// TwinCAT 3 PLC project mobject_led
// Title: mobject-led
// Company: mobject
// Author: mobject-dev-team
// ProjectVersion: 0.1.1
// ProgramVersion: 3.1.4024.0
// libraries:
//   mobject-core, * (mobject)
//   Tc2_System, * (Beckhoff Automation GmbH)
// project tree:
//   Animation/ ArrayStoredAnimation.TcPOU
//   _Internal/DisplayBuffer/ I_ReadableDisplayBuffer.TcIO, I_WritableDisplayBuffer.TcIO
//   _Internal/Display/ I_Display.TcIO
//   _Internal/GraphicalElement/ I_GraphicalElement.TcIO
//   _Internal/Hardware/EL2574/DUT/ EL2574_ChannelExtendedModePdo.TcDUT, EL2574_ChannelExtendedModePdo_I.TcDUT, EL2574_ChannelExtendedModePdo_I_Status.TcDUT, EL2574_ChannelExtendedModePdo_O.TcDUT, EL2574_ChannelExtendedModePdo_O_ExtendedControl.TcDUT, EL2574_ChannelExtendedModePdo_O_ExtendedControl_Segment.TcDUT
//   _Internal/LedDevice/Interface/ I_LedDevice.TcIO
//   _Internal/LedDevice/ LedDevice.TcPOU
//   _Internal/LedDevice/Null/ NullLedDevice.TcPOU
//   _Internal/PixelFormat/ E_PixelFormat.TcDUT
//   _Internal/Pixel/ Pixel.TcDUT
//   _Internal/Scene/ I_Scene.TcIO
//   _Internal/Symbols/Interface/ I_MonoSymbol.TcIO, I_Symbol.TcIO
//   _Internal/Symbols/ Mono_16x16.TcPOU
//   DisplayBuffer/ DisplayBuffer.TcPOU
//   Hardware/EL2574/ EL2574_ChannelExtendedMode.TcPOU
//   Hardware/Matrix/ LedMatrix.TcPOU
//   / PixelColors.TcGVL
//   Scene/ Scene.TcPOU
//   Symbols/Mono_16x16/ Mono_16x16_Alarm.TcPOU, Mono_16x16_BrakeWarning.TcPOU, Mono_16x16_CircleExclamation.TcPOU, Mono_16x16_DownArrow.TcPOU, Mono_16x16_LeftArrow.TcPOU, Mono_16x16_Play.TcPOU, Mono_16x16_RightArrow.TcPOU, Mono_16x16_Smile.TcPOU, Mono_16x16_Temperature.TcPOU, Mono_16x16_TemperatureDown.TcPOU, Mono_16x16_TemperatureUp.TcPOU, Mono_16x16_UpArrow.TcPOU, Mono_16x16_User.TcPOU

// ---- _Internal/Hardware/EL2574/DUT/EL2574_ChannelExtendedModePdo.TcDUT
{attribute 'GUID' := 'B00DF5E7-F5C8-8EB2-0747-F6A66456AF18'}
{attribute 'pack_mode' := '1'}
TYPE EL2574_ChannelExtendedModePdo :
STRUCT
		{attribute 'GUID' := 'B00DF5E8-F5C8-8EB2-0747-F6A66456AF18'}
		Input AT %I* : EL2574_ChannelExtendedModePdo_I;
		{attribute 'GUID' := 'B00DF5E9-F5C8-8EB2-0747-F6A66456AF18'}
		Output AT %Q* : EL2574_ChannelExtendedModePdo_O;
	END_STRUCT
END_TYPE

// ---- _Internal/Hardware/EL2574/DUT/EL2574_ChannelExtendedModePdo_I.TcDUT
{attribute 'GUID' := 'B00DF5E8-F5C8-8EB2-0747-F6A66456AF18'}
TYPE EL2574_ChannelExtendedModePdo_I :
	STRUCT
		{attribute 'GUID' := '979B0B75-C706-0116-3B7C-F1DA38D9DB6C'}
		Status : EL2574_ChannelExtendedModePdo_I_Status;
		{attribute 'hide'}
		_reserved1 : ARRAY [1..32] OF USINT;
	END_STRUCT
END_TYPE

// ---- _Internal/Hardware/EL2574/DUT/EL2574_ChannelExtendedModePdo_I_Status.TcDUT
{attribute 'GUID' := '979B0B75-C706-0116-3B7C-F1DA38D9DB6C'}
TYPE EL2574_ChannelExtendedModePdo_I_Status :
	STRUCT
		Busy : BIT;
		Transmit : BIT;
		Send_Acknowledge : BIT;
		Update_Acknowledge : BIT;
		Command_Acknowledge : BIT;
		Command_Reject : BIT;
		 {attribute 'hide'}
		_reserved1 : BIT;
		 {attribute 'hide'}
		_reserved2 : BIT;
		 {attribute 'hide'}
		_reserved3 : BIT;
		 {attribute 'hide'}
		_reserved4 : BIT;
		Warning : BIT;
		Error : BIT;
		 {attribute 'hide'}
		_reserved5 : BIT;
		 {attribute 'hide'}
		_reserved6 : BIT;
		 {attribute 'GUID' := '18071995-0000-0000-0000-000000000010}
		Input_Cycle_Counter_Bit0 : BIT;
		 {attribute 'GUID' := '18071995-0000-0000-0000-000000000010}
		Input_Cycle_Counter_Bit1 : BIT;
	END_STRUCT
END_TYPE

// ---- _Internal/Hardware/EL2574/DUT/EL2574_ChannelExtendedModePdo_O.TcDUT
{attribute 'GUID' := 'B00DF5E9-F5C8-8EB2-0747-F6A66456AF18'}
{attribute 'pack_mode' := '1'}
TYPE EL2574_ChannelExtendedModePdo_O :
	STRUCT
		 {attribute 'GUID' := 'FCFFC25C-7C92-C549-757B-D5CF9395F3F6'}
		ExtendedControl : EL2574_ChannelExtendedModePdo_O_ExtendedControl;
	END_STRUCT
END_TYPE

// ---- _Internal/Hardware/EL2574/DUT/EL2574_ChannelExtendedModePdo_O_ExtendedControl.TcDUT
{attribute 'GUID' := 'FCFFC25C-7C92-C549-757B-D5CF9395F3F6'}
{attribute 'pack_mode' := '1'}
TYPE EL2574_ChannelExtendedModePdo_O_ExtendedControl :
	STRUCT
		Execute : BIT;
		Send : BIT;
		Update : BIT;
		Write : BIT;
		 {attribute 'hide'}
		_reserved1 : BIT;
		 {attribute 'hide'}
		_reserved2 : BIT;
		 {attribute 'hide'}
		_reserved3 : BIT;
		 {attribute 'hide'}
		_reserved4 : BIT;
		Index : USINT;
		 {attribute 'GUID' := 'C34ECFC1-C235-2097-8F87-A8742B490E4F'}
		Segment : EL2574_ChannelExtendedModePdo_O_ExtendedControl_Segment;
	END_STRUCT
END_TYPE

// ---- _Internal/Hardware/EL2574/DUT/EL2574_ChannelExtendedModePdo_O_ExtendedControl_Segment.TcDUT
{attribute 'GUID' := 'C34ECFC1-C235-2097-8F87-A8742B490E4F'}
TYPE EL2574_ChannelExtendedModePdo_O_ExtendedControl_Segment :
	STRUCT
		Element_0 : UDINT;
		Element_1 : UDINT;
		Element_2 : UDINT;
		Element_3 : UDINT;
		Element_4 : UDINT;
		Element_5 : UDINT;
		Element_6 : UDINT;
		Element_7 : UDINT;
	END_STRUCT
END_TYPE

// ---- _Internal/PixelFormat/E_PixelFormat.TcDUT
{attribute 'qualified_only'}
{attribute 'strict'}
TYPE E_PixelFormat :
(
	RRGGBBAA,
	AARRGGBB,
	xxRRGGBB
);
END_TYPE

// ---- _Internal/Pixel/Pixel.TcDUT
TYPE Pixel : UDINT; END_TYPE

// ---- PixelColors.TcGVL
{attribute 'qualified_only'}
VAR_GLOBAL CONSTANT;
	RED : Pixel := 16#FF0000FF;
	GREEN : Pixel := 16#00FF00FF;
	BLUE : Pixel := 16#0000FFFF;
	YELLOW : Pixel := 16#FFFF00FF;
	BLACK : Pixel := 16#000000FF;
	WHITE : Pixel := 16#FFFFFFF;
	PURPLE : Pixel := 16#800080FF;
	ORANGE : Pixel := 16#FFA500FF;
	GREY : Pixel := 16#808080FF;
	TEAL : Pixel := 16#008080FF;
	CYAN : Pixel := 16#00FFFFF;
	MAGENTA : Pixel := 16#FF00FFFF;
	LIME : Pixel := 16#00FF00FF;
	PINK : Pixel := 16#FFC0CBFF;
	BROWN : Pixel := 16#A52A2AFF;
	NAVY : Pixel := 16#000080FF;
	OLIVE : Pixel := 16#808000FF;
	MAROON : Pixel := 16#800000FF;
	AQUA : Pixel := 16#00FFFFF;
END_VAR

// ---- _Internal/DisplayBuffer/I_ReadableDisplayBuffer.TcIO
INTERFACE I_ReadableDisplayBuffer

METHOD PUBLIC TryReadPixel : BOOL;
VAR_INPUT
	X : DINT;
	Y : DINT;
	Pixel : REFERENCE TO Pixel;
END_VAR
END_METHOD

END_INTERFACE

// ---- _Internal/DisplayBuffer/I_WritableDisplayBuffer.TcIO
INTERFACE I_WritableDisplayBuffer

METHOD PUBLIC SetPixel
VAR_INPUT
	X : DINT;
	Y : DINT;
	Pixel : Pixel;
END_VAR
END_METHOD

END_INTERFACE

// ---- _Internal/Display/I_Display.TcIO
INTERFACE I_Display

METHOD PUBLIC UpdateFrom
VAR_INPUT
	Source : I_ReadableDisplayBuffer;
END_VAR
END_METHOD

END_INTERFACE

// ---- _Internal/GraphicalElement/I_GraphicalElement.TcIO
INTERFACE I_GraphicalElement

METHOD PUBLIC RenderTo
VAR_INPUT
	Destination : I_WritableDisplayBuffer;
END_VAR
END_METHOD

METHOD PUBLIC Update
VAR_INPUT
	DeltaTimeInMs : UDINT;
END_VAR
END_METHOD

END_INTERFACE

// ---- _Internal/LedDevice/Interface/I_LedDevice.TcIO
INTERFACE I_LedDevice EXTENDS I_Display

METHOD PUBLIC ConnectTo
VAR_INPUT
	LedDevice : I_LedDevice;
END_VAR
END_METHOD

METHOD PUBLIC ResetPixelPointer
VAR_INPUT
END_VAR
END_METHOD

METHOD PUBLIC TryGetNextPixel : BOOL
VAR_INPUT
	Destination : REFERENCE TO Pixel;
END_VAR
END_METHOD

METHOD PUBLIC UpdateFrom
VAR_INPUT
	Source : I_ReadableDisplayBuffer;
END_VAR
END_METHOD

END_INTERFACE

// ---- _Internal/Scene/I_Scene.TcIO
INTERFACE I_Scene EXTENDS I_GraphicalElement

METHOD Clear
VAR_INPUT
END_VAR
END_METHOD

METHOD PUBLIC TryAddElement
VAR_INPUT
	GraphicalElement : I_GraphicalElement;
END_VAR
END_METHOD

METHOD PUBLIC TryRemoveElement
VAR_INPUT
	GraphicalElement : I_GraphicalElement;
END_VAR
END_METHOD

END_INTERFACE

// ---- _Internal/Symbols/Interface/I_MonoSymbol.TcIO
INTERFACE I_MonoSymbol EXTENDS I_Symbol

PROPERTY PUBLIC BackgroundColor : Pixel
GET
END_GET
SET
END_SET
END_PROPERTY

PROPERTY PUBLIC ForgroundColor : Pixel
GET
END_GET
SET
END_SET
END_PROPERTY

METHOD PUBLIC InvertColor
VAR_INPUT
END_VAR
END_METHOD

END_INTERFACE

// ---- _Internal/Symbols/Interface/I_Symbol.TcIO
INTERFACE I_Symbol EXTENDS I_GraphicalElement

PROPERTY PUBLIC FlipX : BOOL
GET
END_GET
SET
END_SET
END_PROPERTY

PROPERTY PUBLIC FlipY : BOOL
GET
END_GET
SET
END_SET
END_PROPERTY

PROPERTY PUBLIC Rotation : UINT
GET
END_GET
SET
END_SET
END_PROPERTY

END_INTERFACE

// ---- Animation/ArrayStoredAnimation.TcPOU
{attribute 'linkalways'} 
{attribute 'no_explicit_call' := 'This FB is a CLASS and must be accessed using methods or properties'}
{attribute 'enable_dynamic_creation'}
FUNCTION_BLOCK ArrayStoredAnimation IMPLEMENTS I_GraphicalElement
VAR
	// setup
	_width : UDINT;
	_height : UDINT;
	
	// buffer
	expectedFrameSizeInBytes : UDINT;
	frameCount : UDINT;
	pAnimationFrameData : POINTER TO Pixel;
	nAnimationFrameData : UDINT;
	
	// animation
	currentFrameIndex : UDINT;
	pCurrentFrame : POINTER TO Pixel;
	elapsedTimeInMs : UDINT;
END_VAR

METHOD FB_exit : BOOL
VAR_INPUT
	bInCopyCode : BOOL; // if TRUE, the exit method is called for exiting an instance that is copied afterwards (online change).
END_VAR
IF bInCopyCode THEN
	RETURN;
END_IF

IF pAnimationFrameData = 0 THEN
	RETURN;
END_IF

__DELETE(pAnimationFrameData);
END_METHOD

METHOD FB_init : BOOL
VAR_INPUT
	bInitRetains : BOOL; // if TRUE, the retain variables are initialized (warm start / cold start)
	bInCopyCode : BOOL;  // if TRUE, the instance afterwards gets moved into the copy code (online change)
	Width : UDINT;
	Height : UDINT;
END_VAR
_width := Width;
_height := Height;
UpdateExpectedFrameSizeInBytes();
END_METHOD

PROPERTY PUBLIC Height : UDINT
GET
Height := _height;
END_GET
END_PROPERTY

METHOD PUBLIC RenderTo
VAR_INPUT
	Destination : I_WritableDisplayBuffer;
END_VAR
// needs implementation

//IF X > _width THEN
//	RETURN;
//END_IF

//IF Y > _height THEN
//	RETURN;
//END_IF

//IF frameCount = 0 THEN
//	RETURN;
//END_IF

//offset := (y * width) + x;
//Destination := pCurrentFrame[offset];
//GetPixel := TRUE;
END_METHOD

METHOD PUBLIC Reset : BOOL
VAR_INPUT
END_VAR
Reset := TryGoToFrame(0);
END_METHOD

METHOD PRIVATE ResetAnimation
VAR_INPUT
END_VAR
currentFrameIndex := 0;
pCurrentFrame := pAnimationFrameData;
END_METHOD

METHOD PUBLIC TryAddFrame : BOOL
VAR_INPUT
	FrameDataArray : ANY;
END_VAR
VAR
	newFrameCount : UDINT;
	newAnimationDataSize : UDINT;
	pNewAnimationFrameData : POINTER TO pixel;
	pNewFrameStart : POINTER TO pixel; 
END_VAR
IF FrameDataArray.pValue = 0 THEN
	RETURN;
END_IF

IF FrameDataArray.diSize = 0 THEN
	RETURN;
END_IF

IF FrameDataArray.diSize <> expectedFrameSizeInBytes THEN
	RETURN;
END_IF

// setup the new buffer (one frame bigger than previous)
newFrameCount := frameCount + 1;
newAnimationDataSize := expectedFrameSizeInBytes * newFrameCount;
pNewAnimationFrameData := __NEW(BYTE, newAnimationDataSize);

// copy the old data across if available;
IF nAnimationFrameData > 0 THEN
	memcpy(pNewAnimationFrameData, pAnimationFrameData, nAnimationFrameData); 
	__DELETE(pAnimationFrameData);
	pAnimationFrameData := 0;
	nAnimationFrameData := 0;
END_IF

// copy the supplied frame data to the end of the new buffer.
pNewFrameStart := pNewAnimationFrameData + (frameCount * expectedFrameSizeInBytes);
memcpy(pNewFrameStart, FrameDataArray.pValue, FrameDataArray.diSize); 

// update internal values to the new values.
pAnimationFrameData := pNewAnimationFrameData;
nAnimationFrameData := newAnimationDataSize;
frameCount := newFrameCount;

// reset animation
ResetAnimation();

// success
TryAddFrame := TRUE;
END_METHOD

METHOD PUBLIC TryGoToFrame : BOOL
VAR_INPUT
	AnimationFrameIndex : UDINT;
END_VAR
IF frameCount = 0 THEN 
	RETURN;
END_IF

IF AnimationFrameIndex > frameCount THEN
	RETURN;
END_IF

currentFrameIndex := AnimationFrameIndex;
pCurrentFrame := pAnimationFrameData + (currentFrameIndex * expectedFrameSizeInBytes);
TryGoToFrame := TRUE;
END_METHOD

METHOD PUBLIC TryGoToNextFrame : BOOL
VAR_INPUT
END_VAR
TryGoToNextFrame := TryGoToFrame(currentFrameIndex + 1);
END_METHOD

METHOD PUBLIC Update
VAR_INPUT
	DeltaTimeInMs : UDINT;
END_VAR
// not implemented
END_METHOD

METHOD PRIVATE UpdateExpectedFrameSizeInBytes
VAR
	tempPixel : Pixel;
END_VAR
expectedFrameSizeInBytes := SIZEOF(tempPixel) * this^._width * this^._height;
END_METHOD

PROPERTY PUBLIC Width : UDINT
GET
Width := _width;
END_GET
END_PROPERTY

END_FUNCTION_BLOCK

// ---- _Internal/LedDevice/LedDevice.TcPOU
{attribute 'linkalways'} 
{attribute 'no_explicit_call' := 'This FB is a CLASS and must be accessed using methods or properties'}
{attribute 'enable_dynamic_creation'}
FUNCTION_BLOCK ABSTRACT LedDevice IMPLEMENTS I_LedDevice
VAR
	// using the null object pattern so that you no longer need to check to see if next is <> 0
	nullLedDevice : NullLedDevice;
	next : I_LedDevice := NullLedDevice;
	allPixelsSerialized : BOOL;
	_requiredPixelFormat : E_PixelFormat := E_PixelFormat.AARRGGBB;
END_VAR

METHOD PUBLIC ConnectTo
VAR_INPUT
	LedDevice : I_LedDevice;
END_VAR
IF LedDevice = 0  THEN
	next := nullLedDevice;
END_IF

IF LedDevice = next THEN
	RETURN;
END_IF

next := LedDevice;
END_METHOD

METHOD PROTECTED Convert_RGBA_To_RequiredPixelFormat : Pixel
VAR_INPUT
	Input : Pixel;
END_VAR
CASE _requiredPixelFormat OF
	E_PixelFormat.RRGGBBAA :
		Convert_RGBA_To_RequiredPixelFormat := Input;
		
	E_PixelFormat.AARRGGBB, 
	E_PixelFormat.xxRRGGBB :
		Convert_RGBA_To_RequiredPixelFormat := ROR(Input,8) ; 
END_CASE
END_METHOD

PROPERTY PUBLIC NextDevice : I_LedDevice
GET
NextDevice := next;
END_GET
END_PROPERTY

METHOD PROTECTED ABSTRACT OnResetPixelPointer
VAR_INPUT
END_VAR
// a serializer will be instructed to reset it's own pixel tracking here. 
// this indicates that the next time OnTryGetNextPixel is called, the first pixel must be returned;
END_METHOD

METHOD PROTECTED ABSTRACT OnTryGetNextPixel : BOOL
VAR_INPUT
	Destination : REFERENCE TO Pixel;
END_VAR
// a serializer must keep track of it's own next pixel and set the destination, and return true when called.  
// if there are no further pixels you must return false
END_METHOD

METHOD PROTECTED ABSTRACT OnUpdateFrom
VAR_INPUT
	Source : I_ReadableDisplayBuffer;
END_VAR
END_METHOD

PROPERTY PUBLIC RequiredPixelFormat : E_PixelFormat
GET
RequiredPixelFormat := _requiredPixelFormat;
END_GET
SET
_requiredPixelFormat := RequiredPixelFormat;
END_SET
END_PROPERTY

METHOD PUBLIC ResetPixelPointer
VAR_INPUT
END_VAR
OnResetPixelPointer();
allPixelsSerialized := FALSE;
NextDevice.ResetPixelPointer();
END_METHOD

METHOD PUBLIC TryGetNextPixel : BOOL
VAR_INPUT
	Destination : REFERENCE TO Pixel;
END_VAR
IF allPixelsSerialized THEN
	TryGetNextPixel := NextDevice.TryGetNextPixel(Destination);
	RETURN;
END_IF

IF OnTryGetNextPixel(Destination) THEN
	TryGetNextPixel := TRUE;
	RETURN;
END_IF

allPixelsSerialized := TRUE;
TryGetNextPixel := NextDevice.TryGetNextPixel(Destination);
END_METHOD

METHOD PUBLIC UpdateFrom
VAR_INPUT
	Source : I_ReadableDisplayBuffer;
END_VAR
IF Source = 0 THEN
	RETURN;
END_IF

OnUpdateFrom(Source);
END_METHOD

END_FUNCTION_BLOCK

// ---- _Internal/LedDevice/Null/NullLedDevice.TcPOU
{attribute 'linkalways'} 
{attribute 'no_explicit_call' := 'This FB is a CLASS and must be accessed using methods or properties'}
{attribute 'enable_dynamic_creation'}
FUNCTION_BLOCK NullLedDevice IMPLEMENTS I_LedDevice
VAR
END_VAR

METHOD PUBLIC ConnectTo
VAR_INPUT
	LedDevice : I_LedDevice;
END_VAR
// no code here..
END_METHOD

METHOD PUBLIC ResetPixelPointer
VAR_INPUT
END_VAR
// no code here..
END_METHOD

METHOD PUBLIC TryGetNextPixel : BOOL
VAR_INPUT
	Destination : REFERENCE TO Pixel;
END_VAR
TryGetNextPixel := FALSE;
END_METHOD

METHOD PUBLIC UpdateFrom
VAR_INPUT
	Source : I_ReadableDisplayBuffer;
END_VAR
// no code here..
END_METHOD

END_FUNCTION_BLOCK

// ---- _Internal/Symbols/Mono_16x16.TcPOU
{attribute 'linkalways'} 
{attribute 'no_explicit_call' := 'This FB is a CLASS and must be accessed using methods or properties'}
{attribute 'enable_dynamic_creation'}
FUNCTION_BLOCK ABSTRACT Mono_16x16 IMPLEMENTS I_MonoSymbol
VAR
	_x : DINT;
	_y : DINT;
	_flipX : BOOL;
	_flipY : BOOL;
	_rotation : UINT;
	_forgroundColor : Pixel := WHITE;
	_backgroundColor : Pixel := TRANSPARENT;
END_VAR
VAR CONSTANT
	SYMBOL_WIDTH : UDINT := 16;
	SYMBOL_HEIGHT : UDINT := 16;
	WHITE : Pixel := 16#FFFFFFFF;
	TRANSPARENT : Pixel := 16#00000000;
END_VAR

PROPERTY PUBLIC BackgroundColor : Pixel
GET
BackgroundColor := _backgroundColor;
END_GET
SET
_backgroundColor := BackgroundColor;
END_SET
END_PROPERTY

METHOD FB_init : BOOL
VAR_INPUT
	bInitRetains : BOOL; // if TRUE, the retain variables are initialized (warm start / cold start)
	bInCopyCode : BOOL;  // if TRUE, the instance afterwards gets moved into the copy code (online change)
	Forground : Pixel;
	Background : Pixel;
END_VAR
_forgroundColor := Forground;
_backgroundColor := Background;
END_METHOD

PROPERTY PUBLIC FlipX : BOOL
GET
FlipX := _flipX;
END_GET
SET
_flipX := FlipX;
END_SET
END_PROPERTY

PROPERTY PUBLIC FlipY : BOOL
GET
FlipY := _flipY;
END_GET
SET
_flipY := FlipY;
END_SET
END_PROPERTY

PROPERTY PUBLIC ForgroundColor : Pixel
GET
ForgroundColor := _forgroundColor;
END_GET
SET
_forgroundColor := ForgroundColor;
END_SET
END_PROPERTY

PROPERTY PUBLIC Height : UDINT
GET
Height := SYMBOL_HEIGHT;
END_GET
END_PROPERTY

METHOD PUBLIC InvertColor
VAR_INPUT
END_VAR
END_METHOD

PROPERTY PROTECTED ABSTRACT Pixels : REFERENCE TO ARRAY [0..255] of BYTE
GET
END_GET
END_PROPERTY

METHOD PUBLIC RenderTo
VAR_INPUT
	Destination : I_WritableDisplayBuffer;
END_VAR
VAR
	row : UDINT;
	column : UDINT;
	newRow : UDINT;
	newColumn : UDINT;
	pixelOffset : UDINT;
	destinationX : DINT;
	destinationY : DINT;
END_VAR
FOR row := 0 TO SYMBOL_HEIGHT - 1 DO
	FOR column := 0 TO SYMBOL_WIDTH - 1 DO

		CASE _rotation OF
			
			0:
				newColumn := column;
				newRow := row;
			90:
				newColumn := SYMBOL_HEIGHT - 1 - row;
				newRow := column;
			180:
				newColumn := SYMBOL_WIDTH - 1 - column;
				newRow := SYMBOL_HEIGHT - 1 - row;
			270:
				newColumn := row;
				newRow := SYMBOL_WIDTH - 1 - column;
			
		END_CASE

		IF _flipX THEN
			newColumn := SYMBOL_WIDTH - 1 - newColumn;
		END_IF

		IF _flipY THEN
			newRow := SYMBOL_HEIGHT - 1 - newRow;
		END_IF

		pixelOffset := (newRow * SYMBOL_WIDTH) + newColumn;
		destinationX := UDINT_TO_DINT(column) + _x;
		destinationY := UDINT_TO_DINT(row) + _y;
		
		IF Pixels[pixelOffset] = 0 THEN
			Destination.SetPixel(destinationX, destinationY, _backgroundColor);
		ELSE
			Destination.SetPixel(destinationX, destinationY, _forgroundColor);
		END_IF

	END_FOR
END_FOR
END_METHOD

PROPERTY PUBLIC Rotation : UINT
GET
Rotation := _rotation;
END_GET
SET
_rotation := Rotation;
END_SET
END_PROPERTY

METHOD PUBLIC Update
VAR_INPUT
	DeltaTimeInMs : UDINT;
END_VAR
// not required for static symbols
END_METHOD

PROPERTY PUBLIC Width : UDINT
GET
Width := SYMBOL_WIDTH;
END_GET
END_PROPERTY

PROPERTY PUBLIC X : DINT
GET
X := _x;
END_GET
SET
_x := X;
END_SET
END_PROPERTY

PROPERTY PUBLIC Y : DINT
GET
Y := _y;
END_GET
SET
_y := Y;
END_SET
END_PROPERTY

END_FUNCTION_BLOCK

// ---- DisplayBuffer/DisplayBuffer.TcPOU
{attribute 'linkalways'} 
{attribute 'no_explicit_call' := 'This FB is a CLASS and must be accessed using methods or properties'}
{attribute 'enable_dynamic_creation'}
FUNCTION_BLOCK DisplayBuffer IMPLEMENTS I_WritableDisplayBuffer, I_ReadableDisplayBuffer
VAR
	// setup
	_width : UDINT;
	_height : UDINT;
	
	// buffer
	displayBufferSize : UDINT;
	pDisplayBuffer : POINTER TO Pixel;
END_VAR

METHOD PUBLIC Clear
VAR_INPUT
END_VAR
IF pDisplayBuffer = 0 THEN
	RETURN;
END_IF

memset(pDisplayBuffer, 0, displayBufferSize);
END_METHOD

METHOD PRIVATE CreateDisplayBuffer
VAR
	tempPixel : Pixel;
END_VAR
displayBufferSize := _width * _height * SIZEOF(tempPixel);
pDisplayBuffer := __NEW(BYTE, displayBufferSize);
memset(pDisplayBuffer, 0, displayBufferSize);
END_METHOD

METHOD FB_exit : BOOL
VAR_INPUT
	bInCopyCode : BOOL; // if TRUE, the exit method is called for exiting an instance that is copied afterwards (online change).
END_VAR
IF bInCopyCode THEN
	RETURN;
END_IF

IF pDisplayBuffer = 0 THEN
	RETURN;
END_IF

__DELETE(pDisplayBuffer);
END_METHOD

METHOD FB_init : BOOL
VAR_INPUT
	bInitRetains : BOOL; // if TRUE, the retain variables are initialized (warm start / cold start)
	bInCopyCode : BOOL;  // if TRUE, the instance afterwards gets moved into the copy code (online change)
	Width : UDINT;
	Height : UDINT;
END_VAR
_width := Width;
_height := Height;
CreateDisplayBuffer();
END_METHOD

PROPERTY PUBLIC Height : UDINT
GET
Height := _height;
END_GET
END_PROPERTY

METHOD PUBLIC SendTo
VAR_INPUT
	Display : I_Display;
END_VAR
Display.UpdateFrom(this^);
END_METHOD

METHOD PUBLIC SetPixel
VAR_INPUT
	X : DINT;
	Y : DINT;
	Pixel : Pixel;
END_VAR
VAR
	xAsUdint : UDINT;
	yAsUdint : UDINT;
	offset : UDINT;
END_VAR
IF X < 0 THEN
	RETURN;
END_IF

IF Y < 0 THEN
	RETURN;
END_IF

xAsUdint := DINT_TO_UDINT(X);
yAsUdint := DINT_TO_UDINT(Y);

IF xAsUdint >= _width THEN
	RETURN;
END_IF

IF yAsUdint >= _height THEN
	RETURN;
END_IF


offset := (yAsUdint * _width) + xAsUdint;

IF offset = 176 THEN
			offset := offset;
		END_IF

		
pDisplayBuffer[offset] := Pixel;
END_METHOD

METHOD PUBLIC TryCopyTo : BOOL
VAR_INPUT
	Destination : ANY;
END_VAR
IF DINT_TO_UDINT(Destination.diSize) < displayBufferSize THEN
	RETURN;
END_IF

memcpy(Destination.pValue, pDisplayBuffer, displayBufferSize);
TryCopyTo := true;
END_METHOD

METHOD PUBLIC TryReadPixel : BOOL;
VAR_INPUT
	X : DINT;
	Y : DINT;
	Pixel : REFERENCE TO Pixel;
END_VAR
VAR
	xAsUdint : UDINT;
	yAsUdint : UDINT;
	offset : UDINT;
END_VAR
IF X < 0 THEN
	RETURN;
END_IF

IF Y < 0 THEN
	RETURN;
END_IF

xAsUdint := DINT_TO_UDINT(X);
yAsUdint := DINT_TO_UDINT(Y);

IF xAsUdint >= _width THEN
	RETURN;
END_IF

IF yAsUdint >= _height THEN
	RETURN;
END_IF

offset := (yAsUdint * _width) + xAsUdint;
Pixel := pDisplayBuffer[offset];
TryReadPixel := TRUE;
END_METHOD

PROPERTY PUBLIC Width : UDINT
GET
Width := _width;
END_GET
END_PROPERTY

END_FUNCTION_BLOCK

// ---- Hardware/EL2574/EL2574_ChannelExtendedMode.TcPOU
{attribute 'linkalways'} 
{attribute 'no_explicit_call' := 'This FB is a CLASS and must be accessed using methods or properties'}
{attribute 'enable_dynamic_creation'}
FUNCTION_BLOCK EL2574_ChannelExtendedMode
VAR
	pdo : EL2574_ChannelExtendedModePdo;
	nullLedDevice : NullLedDevice;
	connectedTo : I_LedDevice := NullLedDevice;
	
	totalPixels : UDINT;
	sendBuffer : ARRAY [0..MAX_PIXELS - 1] OF UDINT;
	sendSegmentCount : USINT;
	currentSegment : USINT;
	state : (IDLE, INITIALIZING, SEND_SEGMENT, TRIGGER_FRAME_SEND, WAIT_FOR_FRAME_SEND_COMPLETE, ERROR);
END_VAR
VAR CONSTANT
	MAX_PIXELS : UDINT := 2048;
END_VAR

METHOD PUBLIC ConnectTo
VAR_INPUT
	LedDevice : I_LedDevice;
END_VAR
IF LedDevice = 0  THEN
	connectedTo := nullLedDevice;
END_IF

IF LedDevice = connectedTo THEN
	RETURN;
END_IF

connectedTo := LedDevice;
END_METHOD

METHOD PUBLIC CyclicCall
VAR_INPUT
END_VAR
VAR
	totalSegments : UDINT;
	currentPixel : UDINT;
	i : UDINT;
END_VAR
CASE state OF
	
	IDLE : 

		IF connectedTo = 0 THEN
			RETURN;
		END_IF
		
		connectedTo.ResetPixelPointer();
		currentPixel := 0;
		
		// fetch the buffer
		WHILE connectedTo.TryGetNextPixel(sendBuffer[currentPixel]) DO
			currentPixel := currentPixel + 1;
		END_WHILE
		
		totalPixels := currentPixel;
		
		// reset the remainder of the buffer
		FOR i := currentPixel + 1 TO MAX_PIXELS -1 DO 
			sendBuffer[i] := 16#0;
		END_FOR
		
		state := INITIALIZING;
		
	ERROR : RETURN;
	
	INITIALIZING :
	
		// initialize local variables
		currentSegment := 0;
		totalSegments := totalPixels / 8;
		sendSegmentCount := UDINT_TO_USINT(totalSegments);
	
		// reset the card to a known state 
		pdo.Output.ExtendedControl.Index := 0;
		pdo.Output.ExtendedControl.Send := FALSE;
		pdo.Output.ExtendedControl.Update := FALSE;
		pdo.Output.ExtendedControl.Write := FALSE;
		pdo.Output.ExtendedControl.Segment.Element_0 := 0;
		pdo.Output.ExtendedControl.Segment.Element_1 := 0;
		pdo.Output.ExtendedControl.Segment.Element_2 := 0;
		pdo.Output.ExtendedControl.Segment.Element_3 := 0;
		pdo.Output.ExtendedControl.Segment.Element_4 := 0;
		pdo.Output.ExtendedControl.Segment.Element_5 := 0;
		pdo.Output.ExtendedControl.Segment.Element_6 := 0;
		pdo.Output.ExtendedControl.Segment.Element_7 := 0;
		
		// start sending....
		state := SEND_SEGMENT;

	SEND_SEGMENT :
		
		pdo.Output.ExtendedControl.Index := currentSegment;
		pdo.Output.ExtendedControl.Segment.Element_0 := sendBuffer[currentSegment * 8 + 0];
		pdo.Output.ExtendedControl.Segment.Element_1 := sendBuffer[currentSegment * 8 + 1];
		pdo.Output.ExtendedControl.Segment.Element_2 := sendBuffer[currentSegment * 8 + 2];
		pdo.Output.ExtendedControl.Segment.Element_3 := sendBuffer[currentSegment * 8 + 3];
		pdo.Output.ExtendedControl.Segment.Element_4 := sendBuffer[currentSegment * 8 + 4];
		pdo.Output.ExtendedControl.Segment.Element_5 := sendBuffer[currentSegment * 8 + 5];
		pdo.Output.ExtendedControl.Segment.Element_6 := sendBuffer[currentSegment * 8 + 6];
		pdo.Output.ExtendedControl.Segment.Element_7 := sendBuffer[currentSegment * 8 + 7];
		pdo.Output.ExtendedControl.Write := TRUE;
		pdo.Output.ExtendedControl.Execute := NOT pdo.Output.ExtendedControl.Execute;
		
		IF currentSegment = sendSegmentCount THEN
			state := TRIGGER_FRAME_SEND;
		ELSE
			currentSegment := currentSegment + 1;
		END_IF
		
	TRIGGER_FRAME_SEND : 
	
		pdo.Output.ExtendedControl.Write := FALSE;
		pdo.Output.ExtendedControl.Update := TRUE;
		pdo.Output.ExtendedControl.Send := TRUE;
		pdo.Output.ExtendedControl.Execute := NOT pdo.Output.ExtendedControl.Execute;
		
		state := WAIT_FOR_FRAME_SEND_COMPLETE;
		
	WAIT_FOR_FRAME_SEND_COMPLETE:
	
		IF NOT pdo.Input.Status.Busy THEN
			pdo.Output.ExtendedControl.Update := FALSE;
			pdo.Output.ExtendedControl.Send := FALSE;
			state := IDLE;
		END_IF

		
END_CASE
END_METHOD

PROPERTY PUBLIC HasError : BOOL
GET
HasError := state = Error;
END_GET
END_PROPERTY

PROPERTY PUBLIC IsBusy : BOOL
GET
IsBusy := not(state = IDLE or_else state = ERROR);
END_GET
END_PROPERTY

END_FUNCTION_BLOCK

// ---- Hardware/Matrix/LedMatrix.TcPOU
{attribute 'linkalways'} 
{attribute 'no_explicit_call' := 'This FB is a CLASS and must be accessed using methods or properties'}
{attribute 'enable_dynamic_creation'}
FUNCTION_BLOCK LedMatrix EXTENDS LedDevice
VAR
	// setup
	height : UDINT;
	width : UDINT;
	x : DINT;
	y : DINT;
	flipX : BOOL;
	flipY : BOOL;
	rotation : UINT;
	
	// buffer
	pixelBufferSize : UDINT;
	pPixelBuffer : POINTER TO Pixel;
	
	// serializer
	nextPixel : UDINT;
END_VAR

METHOD PRIVATE CreatePixelBuffer
VAR
	tempPixel : Pixel;
END_VAR
pixelBufferSize := width * height * SIZEOF(tempPixel);
pPixelBuffer := __NEW(BYTE, pixelBufferSize);
memset(pPixelBuffer, 0, pixelBufferSize);
END_METHOD

METHOD FB_exit : BOOL
VAR_INPUT
	bInCopyCode : BOOL; // if TRUE, the exit method is called for exiting an instance that is copied afterwards (online change).
END_VAR
IF bInCopyCode THEN
	RETURN;
END_IF

IF pPixelBuffer = 0 THEN
	RETURN;
END_IF

__DELETE(pPixelBuffer);
END_METHOD

METHOD FB_init : BOOL
VAR_INPUT
	bInitRetains : BOOL; // if TRUE, the retain variables are initialized (warm start / cold start)
	bInCopyCode : BOOL;  // if TRUE, the instance afterwards gets moved into the copy code (online change)
	Height : UDINT;
	Width : UDINT;
	X : UDINT;
	Y : UDINT;
	FlipX : BOOL;
	FlipY : BOOL;
	Rotation : UINT;
END_VAR
THIS^.height := Height;
THIS^.width := Width;
THIS^.x := X;
THIS^.y := Y;
THIS^.flipX := FlipX;
THIS^.flipY := FlipY;
THIS^.rotation := Rotation;

CreatePixelBuffer();
END_METHOD

METHOD PROTECTED OnResetPixelPointer
VAR_INPUT
END_VAR
nextPixel := 0;
END_METHOD

METHOD PROTECTED OnTryGetNextPixel : BOOL
VAR_INPUT
	Destination : REFERENCE TO Pixel;
END_VAR
IF nextPixel > pixelBufferSize THEN
	OnTryGetNextPixel := FALSE;
	RETURN;
END_IF

IF pixelBufferSize = 0 THEN
	RETURN;
END_IF

Destination := pPixelBuffer[nextPixel];
nextPixel := nextPixel + 1;
OnTryGetNextPixel := TRUE;
END_METHOD

METHOD PROTECTED OnUpdateFrom
VAR_INPUT
	Source : I_ReadableDisplayBuffer;
END_VAR
VAR
	row : UDINT;
	column : UDINT;
	newRow : UDINT;
	newColumn : UDINT;
	destinationX : DINT;
	destinationY : DINT;
	index: UDINT;
	pixelValue : PIXEL;
END_VAR
FOR row := 0 TO height - 1 DO
	FOR column := 0 TO width - 1 DO
		
		// calculate the index of our own buffer which represents the current col and row
		IF row MOD 2 = 1 THEN
			// on an odd row the direction is reversed.
			index := row * width + ((width - 1) - column);
		ELSE
			index := row * width + column;
		END_IF
		
		CASE rotation OF
			
			0:
				newColumn := column;
				newRow := row;
			90:
				newColumn := height - 1 - row;
				newRow := column;
			180:
				newColumn := width - 1 - column;
				newRow := height - 1 - row;
			270:
				newColumn := row;
				newRow := width - 1 - column;
			
		END_CASE

		IF flipX THEN
			newColumn := width - 1 - newColumn;
		END_IF

		IF flipY THEN
			newRow := height - 1 - newRow;
		END_IF

		destinationX := UDINT_TO_DINT(newColumn) + x;
		destinationY := UDINT_TO_DINT(newRow) + y;
		
		IF NOT Source.TryReadPixel(destinationX, destinationY, pixelValue) THEN
			pPixelBuffer[index] := 16#00000000;
			RETURN;
		END_IF
		
		pPixelBuffer[index] := THIS^.Convert_RGBA_To_RequiredPixelFormat(pixelValue);

	END_FOR
END_FOR
END_METHOD

END_FUNCTION_BLOCK

// ---- Scene/Scene.TcPOU
{attribute 'linkalways'} 
{attribute 'no_explicit_call' := 'This FB is a CLASS and must be accessed using methods or properties'}
{attribute 'enable_dynamic_creation'}
FUNCTION_BLOCK Scene
VAR
	animations : Queue;
	elements : Queue;
END_VAR

METHOD PUBLIC AddAnimation
VAR_INPUT
	GraphicalElement : I_GraphicalElement;
END_VAR
elements.Enqueue(GraphicalElement);
END_METHOD

METHOD PUBLIC AddElement
VAR_INPUT
	GraphicalElement : I_GraphicalElement;
END_VAR
elements.Enqueue(GraphicalElement);
END_METHOD

METHOD Clear
VAR_INPUT
END_VAR
elements.Clear();
END_METHOD

METHOD PUBLIC RenderTo
VAR_INPUT
	Destination : I_WritableDisplayBuffer;
END_VAR
VAR
	enumerator : I_ForwardEnumerator;
	element : I_GraphicalElement;
END_VAR
enumerator := elements.GetEnumerator();

WHILE enumerator.MoveNext() DO
	IF enumerator.TryGet(element) THEN
		element.RenderTo(Destination);
	END_IF
END_WHILE

enumerator.Dispose();
END_METHOD

METHOD PUBLIC TryRemoveElement : BOOL
VAR_INPUT
	GraphicalElement : I_GraphicalElement;
END_VAR
TryRemoveElement := elements.TryRemoveItem(GraphicalElement);
END_METHOD

METHOD PUBLIC Update
VAR_INPUT
	DeltaTimeInMs : UDINT;
END_VAR
VAR
	enumerator : I_ForwardEnumerator;
	element : I_GraphicalElement;
END_VAR
enumerator := elements.GetEnumerator();

WHILE enumerator.MoveNext() DO
	IF enumerator.TryGet(element) THEN
		element.Update(DeltaTimeInMs);
	END_IF
END_WHILE

enumerator.Dispose();
END_METHOD

END_FUNCTION_BLOCK

// ---- Symbols/Mono_16x16/Mono_16x16_Alarm.TcPOU
{attribute 'linkalways'} 
{attribute 'no_explicit_call' := 'This FB is a CLASS and must be accessed using methods or properties'}
{attribute 'enable_dynamic_creation'}
FUNCTION_BLOCK Mono_16x16_Alarm EXTENDS Mono_16x16
VAR
	_pixels : ARRAY [0..255] OF BYTE := [
		0, 0, 0, 0, 0, 0, 0, 0, 0, 0, 0, 0, 0, 0, 0, 0,
		0, 0, 0, 1, 0, 0, 0, 0, 0, 0, 0, 0, 1, 0, 0, 0,
		0, 0, 1, 0, 0, 0, 0, 1, 1, 0, 0, 0, 0, 1, 0, 0,
		0, 0, 1, 0, 0, 0, 1, 1, 1, 1, 0, 0, 0, 1, 0, 0,
		0, 0, 0, 0, 0, 1, 1, 1, 1, 1, 1, 0, 0, 0, 0, 0,
		0, 0, 0, 0, 0, 1, 1, 1, 1, 1, 1, 0, 0, 0, 0, 0,
		0, 0, 0, 0, 0, 1, 1, 1, 1, 1, 1, 0, 0, 0, 0, 0,
		0, 0, 0, 0, 0, 1, 1, 1, 1, 1, 1, 0, 0, 0, 0, 0,
		0, 0, 0, 0, 0, 1, 1, 1, 1, 1, 1, 0, 0, 0, 0, 0,
		0, 0, 0, 0, 0, 1, 1, 1, 1, 1, 1, 0, 0, 0, 0, 0,
		0, 0, 0, 0, 1, 1, 1, 1, 1, 1, 1, 1, 0, 0, 0, 0,
		0, 0, 0, 1, 1, 1, 1, 1, 1, 1, 1, 1, 1, 0, 0, 0,
		0, 0, 0, 1, 1, 1, 1, 1, 1, 1, 1, 1, 1, 0, 0, 0,
		0, 0, 0, 0, 0, 0, 0, 0, 0, 0, 0, 0, 0, 0, 0, 0,
		0, 0, 0, 0, 0, 0, 0, 1, 1, 0, 0, 0, 0, 0, 0, 0,
		0, 0, 0, 0, 0, 0, 0, 0, 0, 0, 0, 0, 0, 0, 0, 0
	];
END_VAR

PROPERTY PROTECTED Pixels : REFERENCE TO ARRAY [0..255] of BYTE
GET
Pixels ref= _pixels;
END_GET
END_PROPERTY

END_FUNCTION_BLOCK

// ---- Symbols/Mono_16x16/Mono_16x16_BrakeWarning.TcPOU
{attribute 'linkalways'} 
{attribute 'no_explicit_call' := 'This FB is a CLASS and must be accessed using methods or properties'}
{attribute 'enable_dynamic_creation'}
FUNCTION_BLOCK Mono_16x16_BrakeWarning EXTENDS Mono_16x16
VAR
	_pixels : ARRAY [0..255] OF BYTE := [
		0, 0, 0, 0, 0, 0, 0, 0, 0, 0, 0, 0, 0, 0, 0, 0,
		0, 0, 0, 0, 0, 0, 0, 0, 0, 0, 0, 0, 0, 0, 0, 0,
		0, 0, 1, 1, 0, 0, 0, 0, 0, 0, 0, 0, 1, 1, 0, 0,
		0, 1, 1, 1, 0, 0, 0, 1, 1, 0, 0, 0, 1, 1, 1, 0,
		0, 1, 1, 0, 0, 0, 0, 1, 1, 0, 0, 0, 0, 1, 1, 0,
		1, 1, 0, 0, 0, 0, 0, 1, 1, 0, 0, 0, 0, 0, 1, 1,
		1, 1, 0, 0, 0, 0, 0, 1, 1, 0, 0, 0, 0, 0, 1, 1,
		1, 1, 0, 0, 0, 0, 0, 1, 1, 0, 0, 0, 0, 0, 1, 1,
		1, 1, 0, 0, 0, 0, 0, 1, 1, 0, 0, 0, 0, 0, 1, 1,
		1, 1, 0, 0, 0, 0, 0, 1, 1, 0, 0, 0, 0, 0, 1, 1,
		1, 1, 0, 0, 0, 0, 0, 0, 0, 0, 0, 0, 0, 0, 1, 1,
		0, 1, 1, 0, 0, 0, 0, 1, 1, 0, 0, 0, 0, 1, 1, 0,
		0, 1, 1, 1, 0, 0, 0, 1, 1, 0, 0, 0, 1, 1, 1, 0,
		0, 0, 1, 1, 0, 0, 0, 0, 0, 0, 0, 0, 1, 1, 0, 0,
		0, 0, 0, 0, 0, 0, 0, 0, 0, 0, 0, 0, 0, 0, 0, 0,
		0, 0, 0, 0, 0, 0, 0, 0, 0, 0, 0, 0, 0, 0, 0, 0
	];
END_VAR

PROPERTY PROTECTED Pixels : REFERENCE TO ARRAY [0..255] of BYTE
GET
Pixels ref= _pixels;
END_GET
END_PROPERTY

END_FUNCTION_BLOCK

// ---- Symbols/Mono_16x16/Mono_16x16_CircleExclamation.TcPOU
{attribute 'linkalways'} 
{attribute 'no_explicit_call' := 'This FB is a CLASS and must be accessed using methods or properties'}
{attribute 'enable_dynamic_creation'}
FUNCTION_BLOCK Mono_16x16_CircleExclamation EXTENDS Mono_16x16
VAR
	_pixels : ARRAY [0..255] OF BYTE := [
		0, 0, 0, 0, 0, 1, 1, 1, 1, 1, 1, 0, 0, 0, 0, 0,
		0, 0, 0, 1, 1, 1, 1, 1, 1, 1, 1, 1, 1, 0, 0, 0,
		0, 0, 1, 1, 1, 0, 0, 0, 0, 0, 0, 1, 1, 1, 0, 0,
		0, 1, 1, 1, 0, 0, 0, 1, 1, 0, 0, 0, 1, 1, 1, 0,
		0, 1, 1, 0, 0, 0, 0, 1, 1, 0, 0, 0, 0, 1, 1, 0,
		1, 1, 0, 0, 0, 0, 0, 1, 1, 0, 0, 0, 0, 0, 1, 1,
		1, 1, 0, 0, 0, 0, 0, 1, 1, 0, 0, 0, 0, 0, 1, 1,
		1, 1, 0, 0, 0, 0, 0, 1, 1, 0, 0, 0, 0, 0, 1, 1,
		1, 1, 0, 0, 0, 0, 0, 1, 1, 0, 0, 0, 0, 0, 1, 1,
		1, 1, 0, 0, 0, 0, 0, 1, 1, 0, 0, 0, 0, 0, 1, 1,
		1, 1, 0, 0, 0, 0, 0, 0, 0, 0, 0, 0, 0, 0, 1, 1,
		0, 1, 1, 0, 0, 0, 0, 1, 1, 0, 0, 0, 0, 1, 1, 0,
		0, 1, 1, 1, 0, 0, 0, 1, 1, 0, 0, 0, 1, 1, 1, 0,
		0, 0, 1, 1, 1, 0, 0, 0, 0, 0, 0, 1, 1, 1, 0, 0,
		0, 0, 0, 1, 1, 1, 1, 1, 1, 1, 1, 1, 1, 0, 0, 0,
		0, 0, 0, 0, 0, 1, 1, 1, 1, 1, 1, 0, 0, 0, 0, 0
	];
END_VAR

PROPERTY PROTECTED Pixels : REFERENCE TO ARRAY [0..255] of BYTE
GET
Pixels ref= _pixels;
END_GET
END_PROPERTY

END_FUNCTION_BLOCK

// ---- Symbols/Mono_16x16/Mono_16x16_DownArrow.TcPOU
{attribute 'linkalways'} 
{attribute 'no_explicit_call' := 'This FB is a CLASS and must be accessed using methods or properties'}
{attribute 'enable_dynamic_creation'}
FUNCTION_BLOCK Mono_16x16_DownArrow EXTENDS Mono_16x16
VAR
	_pixels : ARRAY [0..255] OF BYTE := [
		0, 0, 0, 0, 0, 0, 0, 0, 0, 0, 0, 0, 0, 0, 0, 0,
		0, 0, 0, 0, 0, 0, 1, 1, 1, 1, 0, 0, 0, 0, 0, 0,
		0, 0, 0, 0, 0, 0, 1, 1, 1, 1, 0, 0, 0, 0, 0, 0,
		0, 0, 0, 0, 0, 0, 1, 1, 1, 1, 0, 0, 0, 0, 0, 0,
		0, 0, 0, 0, 0, 0, 1, 1, 1, 1, 0, 0, 0, 0, 0, 0,
		0, 0, 0, 0, 0, 0, 1, 1, 1, 1, 0, 0, 0, 0, 0, 0,
		0, 0, 0, 0, 0, 0, 1, 1, 1, 1, 0, 0, 0, 0, 0, 0,
		0, 0, 0, 0, 0, 0, 1, 1, 1, 1, 0, 0, 0, 0, 0, 0,
		0, 0, 0, 0, 0, 0, 1, 1, 1, 1, 0, 0, 0, 0, 0, 0,
		0, 0, 1, 1, 1, 1, 1, 1, 1, 1, 1, 1, 1, 1, 0, 0,
		0, 0, 0, 1, 1, 1, 1, 1, 1, 1, 1, 1, 1, 0, 0, 0,
		0, 0, 0, 0, 1, 1, 1, 1, 1, 1, 1, 1, 0, 0, 0, 0,
		0, 0, 0, 0, 0, 1, 1, 1, 1, 1, 1, 0, 0, 0, 0, 0,
		0, 0, 0, 0, 0, 0, 1, 1, 1, 1, 0, 0, 0, 0, 0, 0,
		0, 0, 0, 0, 0, 0, 0, 1, 1, 0, 0, 0, 0, 0, 0, 0,
		0, 0, 0, 0, 0, 0, 0, 0, 0, 0, 0, 0, 0, 0, 0, 0
	];
END_VAR

PROPERTY PROTECTED Pixels : REFERENCE TO ARRAY [0..255] of BYTE
GET
Pixels ref= _pixels;
END_GET
END_PROPERTY

END_FUNCTION_BLOCK

// ---- Symbols/Mono_16x16/Mono_16x16_LeftArrow.TcPOU
{attribute 'linkalways'} 
{attribute 'no_explicit_call' := 'This FB is a CLASS and must be accessed using methods or properties'}
{attribute 'enable_dynamic_creation'}
FUNCTION_BLOCK Mono_16x16_LeftArrow EXTENDS Mono_16x16
VAR
	_pixels : ARRAY [0..255] OF BYTE := [
		0, 0, 0, 0, 0, 0, 0, 0, 0, 0, 0, 0, 0, 0, 0, 0,
		0, 0, 0, 0, 0, 0, 0, 0, 0, 0, 0, 0, 0, 0, 0, 0,
		0, 0, 0, 0, 0, 0, 1, 0, 0, 0, 0, 0, 0, 0, 0, 0,
		0, 0, 0, 0, 0, 1, 1, 0, 0, 0, 0, 0, 0, 0, 0, 0,
		0, 0, 0, 0, 1, 1, 1, 0, 0, 0, 0, 0, 0, 0, 0, 0,
		0, 0, 0, 1, 1, 1, 1, 0, 0, 0, 0, 0, 0, 0, 0, 0,
		0, 0, 1, 1, 1, 1, 1, 1, 1, 1, 1, 1, 1, 1, 1, 0,
		0, 1, 1, 1, 1, 1, 1, 1, 1, 1, 1, 1, 1, 1, 1, 0,
		0, 1, 1, 1, 1, 1, 1, 1, 1, 1, 1, 1, 1, 1, 1, 0,
		0, 0, 1, 1, 1, 1, 1, 1, 1, 1, 1, 1, 1, 1, 1, 0,
		0, 0, 0, 1, 1, 1, 1, 0, 0, 0, 0, 0, 0, 0, 0, 0,
		0, 0, 0, 0, 1, 1, 1, 0, 0, 0, 0, 0, 0, 0, 0, 0,
		0, 0, 0, 0, 0, 1, 1, 0, 0, 0, 0, 0, 0, 0, 0, 0,
		0, 0, 0, 0, 0, 0, 1, 0, 0, 0, 0, 0, 0, 0, 0, 0,
		0, 0, 0, 0, 0, 0, 0, 0, 0, 0, 0, 0, 0, 0, 0, 0,
		0, 0, 0, 0, 0, 0, 0, 0, 0, 0, 0, 0, 0, 0, 0, 0
	];
END_VAR

PROPERTY PROTECTED Pixels : REFERENCE TO ARRAY [0..255] of BYTE
GET
Pixels ref= _pixels;
END_GET
END_PROPERTY

END_FUNCTION_BLOCK

// ---- Symbols/Mono_16x16/Mono_16x16_Play.TcPOU
{attribute 'linkalways'} 
{attribute 'no_explicit_call' := 'This FB is a CLASS and must be accessed using methods or properties'}
{attribute 'enable_dynamic_creation'}
FUNCTION_BLOCK Mono_16x16_Play EXTENDS Mono_16x16
VAR
	_pixels : ARRAY [0..255] OF BYTE := [
		0, 0, 0, 0, 0, 0, 0, 0, 0, 0, 0, 0, 0, 0, 0, 0,
		0, 0, 0, 0, 0, 0, 0, 0, 0, 0, 0, 0, 0, 0, 0, 0,
		0, 0, 1, 1, 0, 0, 0, 0, 0, 0, 0, 0, 0, 0, 0, 0,
		0, 0, 1, 1, 1, 1, 0, 0, 0, 0, 0, 0, 0, 0, 0, 0,
		0, 0, 1, 1, 1, 1, 1, 1, 0, 0, 0, 0, 0, 0, 0, 0,
		0, 0, 1, 1, 1, 1, 1, 1, 1, 1, 0, 0, 0, 0, 0, 0,
		0, 0, 1, 1, 1, 1, 1, 1, 1, 1, 1, 1, 0, 0, 0, 0,
		0, 0, 1, 1, 1, 1, 1, 1, 1, 1, 1, 1, 1, 1, 0, 0,
		0, 0, 1, 1, 1, 1, 1, 1, 1, 1, 1, 1, 1, 1, 0, 0,
		0, 0, 1, 1, 1, 1, 1, 1, 1, 1, 1, 1, 0, 0, 0, 0,
		0, 0, 1, 1, 1, 1, 1, 1, 1, 1, 0, 0, 0, 0, 0, 0,
		0, 0, 1, 1, 1, 1, 1, 1, 0, 0, 0, 0, 0, 0, 0, 0,
		0, 0, 1, 1, 1, 1, 0, 0, 0, 0, 0, 0, 0, 0, 0, 0,
		0, 0, 1, 1, 0, 0, 0, 0, 0, 0, 0, 0, 0, 0, 0, 0,
		0, 0, 0, 0, 0, 0, 0, 0, 0, 0, 0, 0, 0, 0, 0, 0,
		0, 0, 0, 0, 0, 0, 0, 0, 0, 0, 0, 0, 0, 0, 0, 0
	];
END_VAR

PROPERTY PROTECTED Pixels : REFERENCE TO ARRAY [0..255] of BYTE
GET
Pixels ref= _pixels;
END_GET
END_PROPERTY

END_FUNCTION_BLOCK

// ---- Symbols/Mono_16x16/Mono_16x16_RightArrow.TcPOU
{attribute 'linkalways'} 
{attribute 'no_explicit_call' := 'This FB is a CLASS and must be accessed using methods or properties'}
{attribute 'enable_dynamic_creation'}
FUNCTION_BLOCK Mono_16x16_RightArrow EXTENDS Mono_16x16
VAR
	_pixels : ARRAY [0..255] OF BYTE := [
		0, 0, 0, 0, 0, 0, 0, 0, 0, 0, 0, 0, 0, 0, 0, 0,
		0, 0, 0, 0, 0, 0, 0, 0, 0, 0, 0, 0, 0, 0, 0, 0,
		0, 0, 0, 0, 0, 0, 0, 0, 0, 1, 0, 0, 0, 0, 0, 0,
		0, 0, 0, 0, 0, 0, 0, 0, 0, 1, 1, 0, 0, 0, 0, 0,
		0, 0, 0, 0, 0, 0, 0, 0, 0, 1, 1, 1, 0, 0, 0, 0,
		0, 0, 0, 0, 0, 0, 0, 0, 0, 1, 1, 1, 1, 0, 0, 0,
		0, 1, 1, 1, 1, 1, 1, 1, 1, 1, 1, 1, 1, 1, 0, 0,
		0, 1, 1, 1, 1, 1, 1, 1, 1, 1, 1, 1, 1, 1, 1, 0,
		0, 1, 1, 1, 1, 1, 1, 1, 1, 1, 1, 1, 1, 1, 1, 0,
		0, 1, 1, 1, 1, 1, 1, 1, 1, 1, 1, 1, 1, 1, 0, 0,
		0, 0, 0, 0, 0, 0, 0, 0, 0, 1, 1, 1, 1, 0, 0, 0,
		0, 0, 0, 0, 0, 0, 0, 0, 0, 1, 1, 1, 0, 0, 0, 0,
		0, 0, 0, 0, 0, 0, 0, 0, 0, 1, 1, 0, 0, 0, 0, 0,
		0, 0, 0, 0, 0, 0, 0, 0, 0, 1, 0, 0, 0, 0, 0, 0,
		0, 0, 0, 0, 0, 0, 0, 0, 0, 0, 0, 0, 0, 0, 0, 0,
		0, 0, 0, 0, 0, 0, 0, 0, 0, 0, 0, 0, 0, 0, 0, 0
	];
END_VAR

PROPERTY PROTECTED Pixels : REFERENCE TO ARRAY [0..255] of BYTE
GET
Pixels ref= _pixels;
END_GET
END_PROPERTY

END_FUNCTION_BLOCK

// ---- Symbols/Mono_16x16/Mono_16x16_Smile.TcPOU
{attribute 'linkalways'} 
{attribute 'no_explicit_call' := 'This FB is a CLASS and must be accessed using methods or properties'}
{attribute 'enable_dynamic_creation'}
FUNCTION_BLOCK Mono_16x16_Smile EXTENDS Mono_16x16
VAR
	_pixels : ARRAY [0..255] OF BYTE := [
		0, 0, 0, 0, 0, 1, 1, 1, 1, 1, 1, 0, 0, 0, 0, 0,
		0, 0, 0, 1, 1, 1, 1, 1, 1, 1, 1, 1, 1, 0, 0, 0,
		0, 0, 1, 1, 1, 0, 0, 0, 0, 0, 0, 1, 1, 1, 0, 0,
		0, 1, 1, 1, 0, 0, 0, 0, 0, 0, 0, 0, 1, 1, 1, 0,
		0, 1, 1, 0, 0, 0, 0, 0, 0, 0, 0, 0, 0, 1, 1, 0,
		1, 1, 0, 0, 0, 1, 1, 0, 0, 1, 1, 0, 0, 0, 1, 1,
		1, 1, 0, 0, 0, 1, 1, 0, 0, 1, 1, 0, 0, 0, 1, 1,
		1, 1, 0, 0, 0, 0, 0, 0, 0, 0, 0, 0, 0, 0, 1, 1,
		1, 1, 0, 0, 0, 0, 0, 0, 0, 0, 0, 0, 0, 0, 1, 1,
		1, 1, 0, 0, 1, 0, 0, 0, 0, 0, 0, 1, 0, 0, 1, 1,
		1, 1, 0, 0, 1, 1, 0, 0, 0, 0, 1, 1, 0, 0, 1, 1,
		0, 1, 1, 0, 0, 1, 1, 1, 1, 1, 1, 0, 0, 1, 1, 0,
		0, 1, 1, 1, 0, 0, 0, 0, 0, 0, 0, 0, 1, 1, 1, 0,
		0, 0, 1, 1, 1, 0, 0, 0, 0, 0, 0, 1, 1, 1, 0, 0,
		0, 0, 0, 1, 1, 1, 1, 1, 1, 1, 1, 1, 1, 0, 0, 0,
		0, 0, 0, 0, 0, 1, 1, 1, 1, 1, 1, 0, 0, 0, 0, 0
	];
END_VAR

PROPERTY PROTECTED Pixels : REFERENCE TO ARRAY [0..255] of BYTE
GET
Pixels ref= _pixels;
END_GET
END_PROPERTY

END_FUNCTION_BLOCK

// ---- Symbols/Mono_16x16/Mono_16x16_Temperature.TcPOU
{attribute 'linkalways'} 
{attribute 'no_explicit_call' := 'This FB is a CLASS and must be accessed using methods or properties'}
{attribute 'enable_dynamic_creation'}
FUNCTION_BLOCK Mono_16x16_Temperature EXTENDS Mono_16x16
VAR
	_pixels : ARRAY [0..255] OF BYTE := [
		0, 0, 0, 0, 0, 0, 0, 0, 0, 0, 0, 0, 0, 0, 0, 0,
		0, 0, 0, 0, 0, 1, 1, 0, 0, 0, 0, 0, 0, 0, 0, 0,
		0, 0, 0, 0, 0, 1, 1, 1, 1, 0, 0, 0, 0, 0, 0, 0,
		0, 0, 0, 0, 0, 1, 1, 0, 0, 0, 0, 0, 0, 0, 0, 0,
		0, 0, 0, 0, 0, 1, 1, 0, 0, 0, 0, 0, 0, 0, 0, 0,
		0, 0, 0, 0, 0, 1, 1, 1, 1, 0, 0, 0, 0, 0, 0, 0,
		0, 0, 0, 0, 0, 1, 1, 0, 0, 0, 0, 0, 0, 0, 0, 0,
		0, 0, 0, 0, 0, 1, 1, 0, 0, 0, 0, 0, 0, 0, 0, 0,
		0, 0, 0, 0, 0, 1, 1, 1, 1, 0, 0, 0, 0, 0, 0, 0,
		0, 0, 0, 0, 0, 1, 1, 0, 0, 0, 0, 0, 0, 0, 0, 0,
		0, 0, 0, 0, 0, 1, 1, 0, 0, 0, 0, 0, 0, 0, 0, 0,
		0, 0, 0, 0, 1, 1, 1, 1, 0, 0, 0, 0, 0, 0, 0, 0,
		1, 0, 1, 0, 1, 1, 1, 1, 0, 1, 0, 1, 0, 1, 0, 1,
		0, 1, 0, 0, 1, 1, 1, 1, 0, 0, 1, 0, 1, 0, 1, 0,
		0, 0, 0, 0, 0, 1, 1, 0, 0, 0, 0, 0, 0, 0, 0, 0,
		0, 0, 0, 0, 0, 0, 0, 0, 0, 0, 0, 0, 0, 0, 0, 0
	];
END_VAR

PROPERTY PROTECTED Pixels : REFERENCE TO ARRAY [0..255] of BYTE
GET
Pixels ref= _pixels;
END_GET
END_PROPERTY

END_FUNCTION_BLOCK

// ---- Symbols/Mono_16x16/Mono_16x16_TemperatureDown.TcPOU
{attribute 'linkalways'} 
{attribute 'no_explicit_call' := 'This FB is a CLASS and must be accessed using methods or properties'}
{attribute 'enable_dynamic_creation'}
FUNCTION_BLOCK Mono_16x16_TemperatureDown EXTENDS Mono_16x16
VAR
	_pixels : ARRAY [0..255] OF BYTE := [
		0, 0, 0, 0, 0, 0, 0, 0, 0, 0, 0, 0, 0, 0, 0, 0,
		0, 0, 0, 0, 0, 1, 1, 0, 0, 0, 0, 0, 0, 0, 0, 0,
		0, 0, 0, 0, 0, 1, 1, 1, 1, 0, 0, 0, 1, 0, 0, 0,
		0, 0, 0, 0, 0, 1, 1, 0, 0, 0, 0, 0, 1, 0, 0, 0,
		0, 0, 0, 0, 0, 1, 1, 0, 0, 0, 0, 0, 1, 0, 0, 0,
		0, 0, 0, 0, 0, 1, 1, 1, 1, 0, 0, 0, 1, 0, 0, 0,
		0, 0, 0, 0, 0, 1, 1, 0, 0, 0, 0, 0, 1, 0, 0, 0,
		0, 0, 0, 0, 0, 1, 1, 0, 0, 0, 1, 1, 1, 1, 1, 0,
		0, 0, 0, 0, 0, 1, 1, 1, 1, 0, 0, 1, 1, 1, 0, 0,
		0, 0, 0, 0, 0, 1, 1, 0, 0, 0, 0, 0, 1, 0, 0, 0,
		0, 0, 0, 0, 0, 1, 1, 0, 0, 0, 0, 0, 0, 0, 0, 0,
		0, 0, 0, 0, 1, 1, 1, 1, 0, 0, 0, 0, 0, 0, 0, 0,
		1, 0, 1, 0, 1, 1, 1, 1, 0, 1, 0, 1, 0, 1, 0, 1,
		0, 1, 0, 0, 1, 1, 1, 1, 0, 0, 1, 0, 1, 0, 1, 0,
		0, 0, 0, 0, 0, 1, 1, 0, 0, 0, 0, 0, 0, 0, 0, 0,
		0, 0, 0, 0, 0, 0, 0, 0, 0, 0, 0, 0, 0, 0, 0, 0
	];
END_VAR

PROPERTY PROTECTED Pixels : REFERENCE TO ARRAY [0..255] of BYTE
GET
Pixels ref= _pixels;
END_GET
END_PROPERTY

END_FUNCTION_BLOCK

// ---- Symbols/Mono_16x16/Mono_16x16_TemperatureUp.TcPOU
{attribute 'linkalways'} 
{attribute 'no_explicit_call' := 'This FB is a CLASS and must be accessed using methods or properties'}
{attribute 'enable_dynamic_creation'}
FUNCTION_BLOCK Mono_16x16_TemperatureUp EXTENDS Mono_16x16
VAR
	_pixels : ARRAY [0..255] OF BYTE := [
		0, 0, 0, 0, 0, 0, 0, 0, 0, 0, 0, 0, 0, 0, 0, 0,
		0, 0, 0, 0, 0, 1, 1, 0, 0, 0, 0, 0, 0, 0, 0, 0,
		0, 0, 0, 0, 0, 1, 1, 1, 1, 0, 0, 0, 1, 0, 0, 0,
		0, 0, 0, 0, 0, 1, 1, 0, 0, 0, 0, 1, 1, 1, 0, 0,
		0, 0, 0, 0, 0, 1, 1, 0, 0, 0, 1, 1, 1, 1, 1, 0,
		0, 0, 0, 0, 0, 1, 1, 1, 1, 0, 0, 0, 1, 0, 0, 0,
		0, 0, 0, 0, 0, 1, 1, 0, 0, 0, 0, 0, 1, 0, 0, 0,
		0, 0, 0, 0, 0, 1, 1, 0, 0, 0, 0, 0, 1, 0, 0, 0,
		0, 0, 0, 0, 0, 1, 1, 1, 1, 0, 0, 0, 1, 0, 0, 0,
		0, 0, 0, 0, 0, 1, 1, 0, 0, 0, 0, 0, 1, 0, 0, 0,
		0, 0, 0, 0, 0, 1, 1, 0, 0, 0, 0, 0, 0, 0, 0, 0,
		0, 0, 0, 0, 1, 1, 1, 1, 0, 0, 0, 0, 0, 0, 0, 0,
		1, 0, 1, 0, 1, 1, 1, 1, 0, 1, 0, 1, 0, 1, 0, 1,
		0, 1, 0, 0, 1, 1, 1, 1, 0, 0, 1, 0, 1, 0, 1, 0,
		0, 0, 0, 0, 0, 1, 1, 0, 0, 0, 0, 0, 0, 0, 0, 0,
		0, 0, 0, 0, 0, 0, 0, 0, 0, 0, 0, 0, 0, 0, 0, 0
	];
END_VAR

PROPERTY PROTECTED Pixels : REFERENCE TO ARRAY [0..255] of BYTE
GET
Pixels ref= _pixels;
END_GET
END_PROPERTY

END_FUNCTION_BLOCK

// ---- Symbols/Mono_16x16/Mono_16x16_UpArrow.TcPOU
{attribute 'linkalways'} 
{attribute 'no_explicit_call' := 'This FB is a CLASS and must be accessed using methods or properties'}
{attribute 'enable_dynamic_creation'}
FUNCTION_BLOCK Mono_16x16_UpArrow EXTENDS Mono_16x16
VAR
	_pixels : ARRAY [0..255] OF BYTE := [
		0, 0, 0, 0, 0, 0, 0, 0, 0, 0, 0, 0, 0, 0, 0, 0,
		0, 0, 0, 0, 0, 0, 0, 1, 1, 0, 0, 0, 0, 0, 0, 0,
		0, 0, 0, 0, 0, 0, 1, 1, 1, 1, 0, 0, 0, 0, 0, 0,
		0, 0, 0, 0, 0, 1, 1, 1, 1, 1, 1, 0, 0, 0, 0, 0,
		0, 0, 0, 0, 1, 1, 1, 1, 1, 1, 1, 1, 0, 0, 0, 0,
		0, 0, 0, 1, 1, 1, 1, 1, 1, 1, 1, 1, 1, 0, 0, 0,
		0, 0, 1, 1, 1, 1, 1, 1, 1, 1, 1, 1, 1, 1, 0, 0,
		0, 0, 0, 0, 0, 0, 1, 1, 1, 1, 0, 0, 0, 0, 0, 0,
		0, 0, 0, 0, 0, 0, 1, 1, 1, 1, 0, 0, 0, 0, 0, 0,
		0, 0, 0, 0, 0, 0, 1, 1, 1, 1, 0, 0, 0, 0, 0, 0,
		0, 0, 0, 0, 0, 0, 1, 1, 1, 1, 0, 0, 0, 0, 0, 0,
		0, 0, 0, 0, 0, 0, 1, 1, 1, 1, 0, 0, 0, 0, 0, 0,
		0, 0, 0, 0, 0, 0, 1, 1, 1, 1, 0, 0, 0, 0, 0, 0,
		0, 0, 0, 0, 0, 0, 1, 1, 1, 1, 0, 0, 0, 0, 0, 0,
		0, 0, 0, 0, 0, 0, 1, 1, 1, 1, 0, 0, 0, 0, 0, 0,
		0, 0, 0, 0, 0, 0, 0, 0, 0, 0, 0, 0, 0, 0, 0, 0
	];
END_VAR

PROPERTY PROTECTED Pixels : REFERENCE TO ARRAY [0..255] of BYTE
GET
Pixels ref= _pixels;
END_GET
END_PROPERTY

END_FUNCTION_BLOCK

// ---- Symbols/Mono_16x16/Mono_16x16_User.TcPOU
{attribute 'linkalways'} 
{attribute 'no_explicit_call' := 'This FB is a CLASS and must be accessed using methods or properties'}
{attribute 'enable_dynamic_creation'}
FUNCTION_BLOCK Mono_16x16_User EXTENDS Mono_16x16
VAR
	_pixels : ARRAY [0..255] OF BYTE := [
		0, 0, 0, 0, 0, 0, 0, 0, 0, 0, 0, 0, 0, 0, 0, 0,
		0, 0, 0, 0, 0, 0, 0, 0, 0, 0, 0, 0, 0, 0, 0, 0,
		0, 0, 0, 0, 0, 0, 0, 0, 0, 0, 0, 0, 0, 0, 0, 0,
		0, 0, 0, 0, 0, 0, 1, 1, 1, 1, 0, 0, 0, 0, 0, 0,
		0, 0, 0, 0, 0, 1, 1, 1, 1, 1, 1, 0, 0, 0, 0, 0,
		0, 0, 0, 0, 0, 1, 1, 1, 1, 1, 1, 0, 0, 0, 0, 0,
		0, 0, 0, 0, 0, 1, 1, 1, 1, 1, 1, 0, 0, 0, 0, 0,
		0, 0, 0, 0, 0, 1, 1, 1, 1, 1, 1, 0, 0, 0, 0, 0,
		0, 0, 0, 0, 0, 0, 1, 1, 1, 1, 0, 0, 0, 0, 0, 0,
		0, 0, 0, 0, 0, 0, 0, 0, 0, 0, 0, 0, 0, 0, 0, 0,
		0, 0, 0, 0, 0, 1, 1, 1, 1, 1, 1, 0, 0, 0, 0, 0,
		0, 0, 0, 0, 1, 1, 1, 1, 1, 1, 1, 1, 0, 0, 0, 0,
		0, 0, 0, 1, 1, 1, 1, 1, 1, 1, 1, 1, 1, 0, 0, 0,
		0, 0, 0, 1, 1, 1, 1, 1, 1, 1, 1, 1, 1, 0, 0, 0,
		0, 0, 0, 1, 1, 1, 1, 1, 1, 1, 1, 1, 1, 0, 0, 0,
		0, 0, 0, 1, 1, 1, 1, 1, 1, 1, 1, 1, 1, 0, 0, 0
	];
END_VAR

PROPERTY PROTECTED Pixels : REFERENCE TO ARRAY [0..255] of BYTE
GET
Pixels ref= _pixels;
END_GET
END_PROPERTY

END_FUNCTION_BLOCK
